// Mitsubishi GX Works2 project: b13   PLC: Q02/Q02H

PROGRAM MAIN
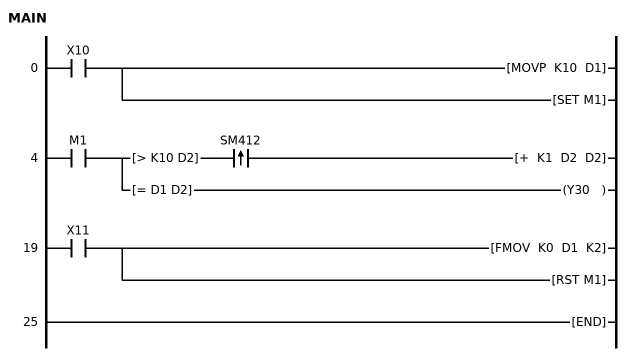
0     LD      X10
      MOVP    K10 D1
      SET     M1
4     LD      M1
      MPS
      AND>    K10 D2
      ANDP    SM412
      +       K1 D2 D2
      MPP
      AND=    D1 D2
      OUT     Y30
19    LD      X11
      FMOV    K0 D1 K2
      RST     M1
25    END
END_PROGRAM
